TYPE ST_AL1333 :
STRUCT
	bStateIOLink				: ARRAY[1..8] OF BOOL;
	nStateIOLink		AT %I*	: ARRAY[1..8] OF USINT;
	bQualifierIOLink 			: ARRAY[1..8] OF BOOL;
	nQualifierIOLink 	AT %I*	: ARRAY[1..8] OF USINT;
END_STRUCT
END_TYPE

(* stored: Version 1.1.0.1, ProductVersion 3.1.4024.12
   DUT ST_AL1333: Id {0459e445-fa05-43e7-b6b2-b44366494b39} *)
